PROGRAM P1_03_MachineControl
VAR
	tonStarting		:TON;
	tonStopping		:TON;
END_VAR

VAR PERSISTENT
	bBatchConfirmation1			:BOOL;
	bBatchConfirmation2			:BOOL;
	bBatchConfirmation3			:BOOL;
	bBatchConfirmation4			:BOOL;
END_VAR
VAR // added by the converter: edge detectors and wires of the graphical bodies
    _w1, _w2, _w3, _w4, _w5, _w6, _w7, _w8, _w9, _w10 : BOOL;
    _rt1, _rt2 : R_TRIG;
END_VAR

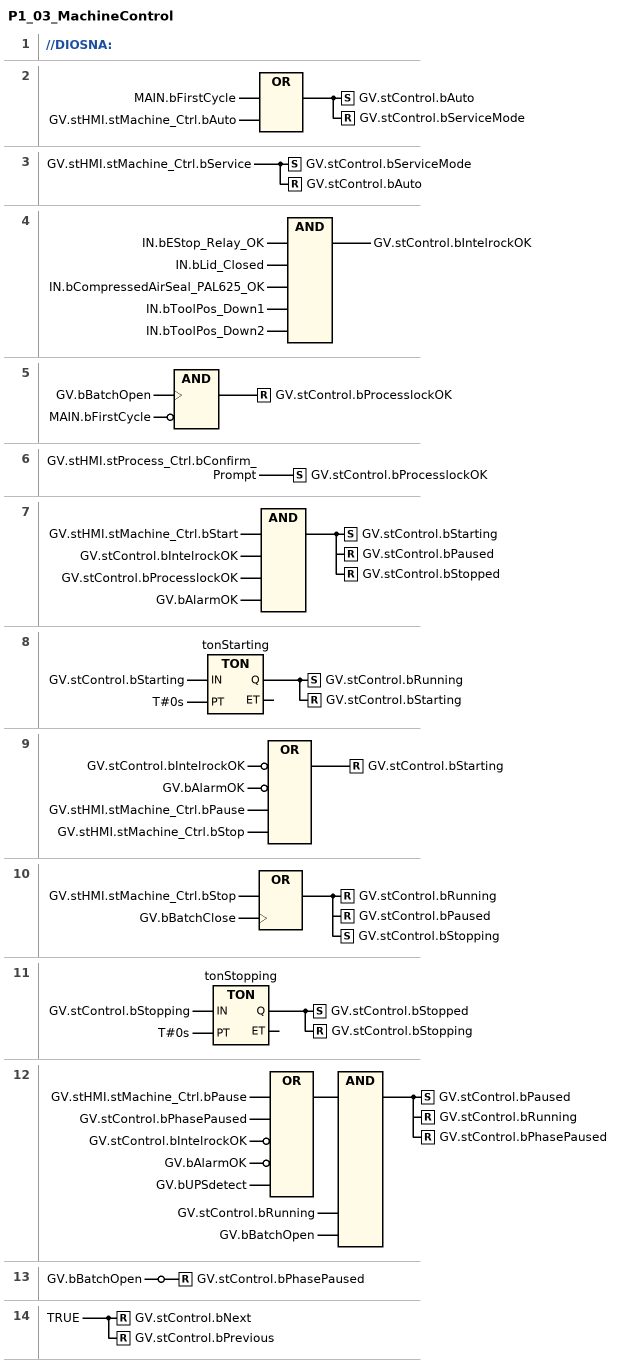
// NETWORK 1
// label: //DIOSNA

// NETWORK 2
_w1 := MAIN.bFirstCycle OR GV.stHMI.stMachine_Ctrl.bAuto;
GV.stControl.bAuto S= _w1;
GV.stControl.bServiceMode R= _w1;

// NETWORK 3
_w2 := GV.stHMI.stMachine_Ctrl.bService;
GV.stControl.bServiceMode S= _w2;
GV.stControl.bAuto R= _w2;

// NETWORK 4
GV.stControl.bIntelrockOK := IN.bEStop_Relay_OK AND IN.bLid_Closed AND IN.bCompressedAirSeal_PAL625_OK AND IN.bToolPos_Down1 AND IN.bToolPos_Down2;

// NETWORK 5
_rt1(CLK := GV.bBatchOpen);
GV.stControl.bProcesslockOK R= _rt1.Q AND NOT MAIN.bFirstCycle;

// NETWORK 6
GV.stControl.bProcesslockOK S= GV.stHMI.stProcess_Ctrl.bConfirm_Prompt;

// NETWORK 7
_w3 := GV.stHMI.stMachine_Ctrl.bStart AND GV.stControl.bIntelrockOK AND GV.stControl.bProcesslockOK AND GV.bAlarmOK;
GV.stControl.bStarting S= _w3;
GV.stControl.bPaused R= _w3;
GV.stControl.bStopped R= _w3;

// NETWORK 8
tonStarting(IN := GV.stControl.bStarting, PT := T#0s); // TON
GV.stControl.bRunning S= tonStarting.Q;
GV.stControl.bStarting R= tonStarting.Q;

// NETWORK 9
GV.stControl.bStarting R= NOT GV.stControl.bIntelrockOK OR NOT GV.bAlarmOK OR GV.stHMI.stMachine_Ctrl.bPause OR GV.stHMI.stMachine_Ctrl.bStop;

// NETWORK 10
_rt2(CLK := GV.bBatchClose);
_w4 := GV.stHMI.stMachine_Ctrl.bStop OR _rt2.Q;
GV.stControl.bRunning R= _w4;
GV.stControl.bPaused R= _w4;
GV.stControl.bStopping S= _w4;

// NETWORK 11
tonStopping(IN := GV.stControl.bStopping, PT := T#0s); // TON
GV.stControl.bStopped S= tonStopping.Q;
GV.stControl.bStopping R= tonStopping.Q;

// NETWORK 12
_w5 := (GV.stHMI.stMachine_Ctrl.bPause OR GV.stControl.bPhasePaused OR NOT GV.stControl.bIntelrockOK OR NOT GV.bAlarmOK OR GV.bUPSdetect) AND GV.stControl.bRunning AND GV.bBatchOpen;
GV.stControl.bPaused S= _w5;
GV.stControl.bRunning R= _w5;
GV.stControl.bPhasePaused R= _w5;

// NETWORK 13
GV.stControl.bPhasePaused R= NOT GV.bBatchOpen;

// NETWORK 14
GV.stControl.bNext R= TRUE;
GV.stControl.bPrevious R= TRUE;

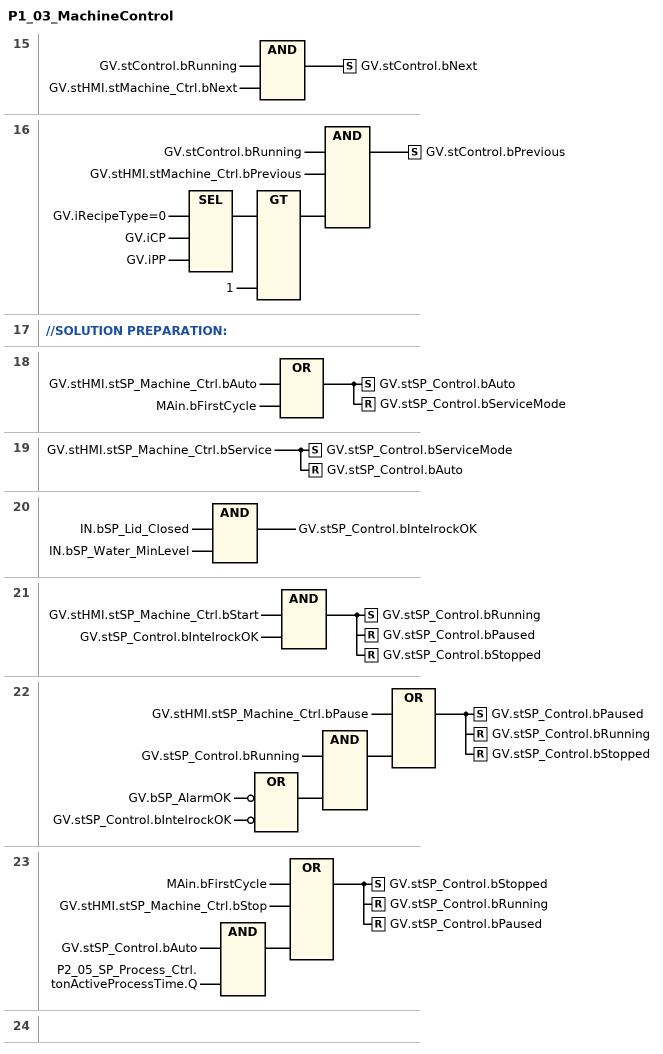
// NETWORK 15
GV.stControl.bNext S= GV.stControl.bRunning AND GV.stHMI.stMachine_Ctrl.bNext;

// NETWORK 16
GV.stControl.bPrevious S= GV.stControl.bRunning AND GV.stHMI.stMachine_Ctrl.bPrevious AND SEL(GV.iRecipeType=0, GV.iCP, GV.iPP) > 1;

// NETWORK 17
// label: //SOLUTION PREPARATION

// NETWORK 18
_w6 := GV.stHMI.stSP_Machine_Ctrl.bAuto OR MAin.bFirstCycle;
GV.stSP_Control.bAuto S= _w6;
GV.stSP_Control.bServiceMode R= _w6;

// NETWORK 19
_w7 := GV.stHMI.stSP_Machine_Ctrl.bService;
GV.stSP_Control.bServiceMode S= _w7;
GV.stSP_Control.bAuto R= _w7;

// NETWORK 20
GV.stSP_Control.bIntelrockOK := IN.bSP_Lid_Closed AND IN.bSP_Water_MinLevel;

// NETWORK 21
_w8 := GV.stHMI.stSP_Machine_Ctrl.bStart AND GV.stSP_Control.bIntelrockOK;
GV.stSP_Control.bRunning S= _w8;
GV.stSP_Control.bPaused R= _w8;
GV.stSP_Control.bStopped R= _w8;

// NETWORK 22
_w9 := GV.stHMI.stSP_Machine_Ctrl.bPause OR GV.stSP_Control.bRunning AND (NOT GV.bSP_AlarmOK OR NOT GV.stSP_Control.bIntelrockOK);
GV.stSP_Control.bPaused S= _w9;
GV.stSP_Control.bRunning R= _w9;
GV.stSP_Control.bStopped R= _w9;

// NETWORK 23
_w10 := MAin.bFirstCycle OR GV.stHMI.stSP_Machine_Ctrl.bStop OR GV.stSP_Control.bAuto AND P2_05_SP_Process_Ctrl.tonActiveProcessTime.Q;
GV.stSP_Control.bStopped S= _w10;
GV.stSP_Control.bRunning R= _w10;
GV.stSP_Control.bPaused R= _w10;

// NETWORK 24

END_PROGRAM

(* stored: Version 1.1.0.1, ProductVersion 3.1.4026.13
   POU P1_03_MachineControl: Id {28291006-7217-4dfd-bae8-40d23c5c0960}, SpecialFunc None *)
